INTERFACE I_Label EXTENDS I_Blank

PROPERTY name : STRING
GET
END_GET
END_PROPERTY

END_INTERFACE

(* stored: Version 1.1.0.1, ProductVersion 3.1.4024.12
   Itf I_Label: Id {3918297b-74d6-4271-b179-36e28f22d825}
   Property name: Id {aefa095b-bbbe-4e22-bf45-965c5a14f3c6}
   Get Get: Id {ad8623f9-ce34-4fda-9da0-32644c497693} *)
